(* IEC 61131-3 sources: CodesysTest/export/Unused/FB_SimBasicBagDelivery.pou/ReadyForPrint.prop, 1 file *)

(* ---- Get.pm.st ---- *)
(*#-#-#-#-#-#-#-#-#-#---Declaration---#-#-#-#-#-#-#-#-#-#-#-#-#*)

VAR
END_VAR
(*#-#-#-#-#-#-#-#-#-#---Implementation---#-#-#-#-#-#-#-#-#-#-#-#-#*)

ReadyForPrint := feedToPrintOffset.Q;
